# EPICS autosave request: soft_iocs/galil_DMC_A01/iocBoot/iocgalil_DMC_A01/GalilTest_18ID_DMC_A01Positions.req
$(P)A1.DVAL
$(P)A2.DVAL
$(P)A3.DVAL
$(P)A4.DVAL
$(P)A5.DVAL
$(P)A6.DVAL
$(P)A7.DVAL
$(P)A8.DVAL
